Universal Robots PolyScope program: example-1.urp

Program example-1 (installation=default directory=/home/ur/ursim/ursim-5.5.1.82186/programs createdIn=5.5.1.82186 lastSavedIn=5.5.1.82186 robotSerialNumber=20183599999)
Calibrated DH parameters: a=[0, -0.425, -0.3922, 0, 0, 0]; d=[0.1625, 0, 0, 0.1333, 0.0997, 0.0996]; alpha=[1.570796, 0, 0, 1.570796, -1.570796, 0]; deltaTheta=[0, 0, 0, 0, 0, 0]
Robot Program (runOnlyOnce=false)
  MoveJ speed 60 deg/s, acceleration 80 deg/s^2 (useActiveTCP=true) feature=Base
    Waypoint Waypoint_1: TCP in base x=-143.969 y=-435.62 z=202.03 mm, rx=-0.0012 ry=3.1163 rz=0.0389 rad; joints [-91.713, -98.956, -126.223, -46.295, 91.392, -1.776] deg
    Waypoint Waypoint_2: TCP in base x=-28.459 y=-432.401 z=318.301 mm, rx=-0.4209 ry=3.0405 rz=-0.3724 rad; joints [-76.186, -83.428, -126.223, -46.295, 91.392, -1.776] deg
    Waypoint Waypoint_1: TCP in base x=-143.969 y=-435.62 z=202.03 mm, rx=-0.0012 ry=3.1163 rz=0.0389 rad; joints [-91.713, -98.956, -126.223, -46.295, 91.392, -1.776] deg
Thread Thread_1 (runOnlyOnce=false)
  Wait Sleep waitTime=0.5
  Script: i_var_1 = get_target_tcp_pose()
  URCap Webservice (NAST Webservice, NAST Automation) dataModel(Variable(key=selectedVar, variable=i_var_1))
